// The read model. Implemented by a suite, and by a sequencer aggregating suites -
// which is what makes sequencers nest and lets a consumer poll one symbol
// regardless of how many suites exist.
//
// Read-only, and separate from the driving surface on purpose: something that only
// wants to know whether the run finished should not also be handed the ability to
// restart it.
//
// Computing all of this every scan and exposing none of it is the trap. The counts
// were private and absent from any interface, so nothing could ask whether a run
// had finished - the only signals were a file appearing on disk and a line in a
// log, both of which have to be scraped.
//
// A flat struct carrying the same values is published alongside, so ADS, TwinCAT
// HMI and OPC UA read it as plain symbols without RPC. That is the portable path,
// and the one CI polls.
INTERFACE I_TestRunStatus EXTENDS I_Labelled

// Tests that could not run, plus framework errors. Kept apart from FailedCount
// because a build should react differently: a failure means the code is wrong, an
// error means the run cannot be trusted.
PROPERTY ErrorCount : UDINT
GET
END_GET
END_PROPERTY

// Checks that did not hold.
PROPERTY FailedCount : UDINT
GET
END_GET
END_PROPERTY

// Reached a terminal state - NOT 'ran everything'.
//
// A skipped suite reports complete. If it did not, any aggregate containing one
// would wait for it forever.
PROPERTY IsComplete : BOOL
GET
END_GET
END_PROPERTY

// Readable while the run is in progress, not only at the end: Outcome
// distinguishes Running from every terminal value.
PROPERTY Outcome : E_RunOutcome
GET
END_GET
END_PROPERTY

PROPERTY PassedCount : UDINT
GET
END_GET
END_PROPERTY

// Not a failure. Must not turn a build red.
PROPERTY SkippedCount : UDINT
GET
END_GET
END_PROPERTY

// Tests registered. Once complete, Passed + Failed + Errored + Skipped equals it.
PROPERTY TestCount : UDINT
GET
END_GET
END_PROPERTY

// Seconds for the whole run: a suite sums its tests, a sequencer sums its
// suites.
//
// Named apart from I_TestTiming.ElapsedTime deliberately. The two are not one
// concept declared twice - one is how long a single test has been going, the
// other an aggregate over many. Two interfaces declaring the same member is a
// design error even when the types match, and here the meanings differ too.
PROPERTY TotalDuration : LREAL
GET
END_GET
END_PROPERTY

END_INTERFACE

(* stored: Version 1.1.0.1, ProductVersion 3.1.4026.18
   Itf I_TestRunStatus: Id {c8fc3484-8a44-4188-ab19-c846b99d133b}
   Property ErrorCount: Id {c138f240-399f-4f01-af72-fcc145dd94ba}
   Get Get: Id {9626a572-8a18-4b74-9afd-531c0ef18442}
   Property FailedCount: Id {7dee69bd-7c13-4d7f-b406-a9609c7fa41e}
   Get Get: Id {65626a81-4f23-4c04-98c0-70881c4c080d}
   Property IsComplete: Id {b4347bcd-2013-432d-8a4b-b20e2a29e5d6}
   Get Get: Id {95d0781c-b9c8-46e7-8b2a-7ca8e9460ec5}
   Property Outcome: Id {8892a887-c10e-4dd4-aced-f9ca9adacf43}
   Get Get: Id {9a60f19a-cd2d-4dd3-9413-4a7a171de037}
   Property PassedCount: Id {69cb7edf-3d83-4d32-bd39-0287b6d763c1}
   Get Get: Id {ebd7237c-5d78-4882-905c-9a524f8edc96}
   Property SkippedCount: Id {91317776-f74d-4eba-965d-91662da5b08a}
   Get Get: Id {8bd1b763-6c91-4f0f-b5b5-c84271286fbd}
   Property TestCount: Id {7ebbfb87-7093-4afa-85db-5d48e51aef1c}
   Get Get: Id {a2b6040a-8e34-495d-b50e-4e5a59663925}
   Property TotalDuration: Id {5b22496c-7227-498a-90d6-dbb9729e135c}
   Get Get: Id {ee62fec0-dd92-4cf5-91aa-251665d4b065} *)
